INTERFACE ICompositeDevice EXTENDS IDevice

{attribute 'monitoring' := 'call'}
PROPERTY SubDeviceCount : INT
GET
END_GET
END_PROPERTY

METHOD TryGetSubDeviceByIndex : IDevice
VAR_INPUT
	index : BYTE;
END_VAR
END_METHOD

END_INTERFACE

(* stored: Version 1.1.0.1
   Itf ICompositeDevice: Id {be5e3b3f-f46a-4c0b-a57f-a0e8cfdaef93}
   Property SubDeviceCount: Id {91c58717-a1a6-455a-8953-051494694324}
   Get Get: Id {b945543f-043e-4a1a-a716-c1a6bb5d5ca0}
   Method TryGetSubDeviceByIndex: Id {ae022ef2-87e5-46a0-ae9e-d3ac431e6e2f} *)
